TYPE ST_FSoE_12Byte :
STRUCT
	CMD		: BYTE;
	SafeData1 	: WORD;
	CRC1		: WORD;
	SafeData2 	: WORD;
	CRC2		: WORD;
	SafeData3 	: WORD;
	CRC3		: WORD;
	SafeData4 	: WORD;
	CRC4		: WORD;
	SafeData5 	: WORD;
	CRC5		: WORD;
	SafeData6 	: WORD;
	CRC6		: WORD;
	ConnID		: WORD;
END_STRUCT
END_TYPE

(* stored: Version 1.1.0.1, ProductVersion 3.1.4024.5
   DUT ST_FSoE_12Byte: Id {86f4f2f2-42d9-4ac1-9c38-7c979bd8abed} *)
